(* IEC 61131-3 sources: RL_MAR/experiments/comparison/llm4plc/results/deepseek-ai-DeepSeek-V3.2_20260506_104945/20260506_110207, 3 files *)

(* ---- generated_code_iteration_0.st ---- *)
START_ST
FUNCTION_BLOCK FB_HexDigitAnalyzer
VAR_INPUT
    InputNumber : INT;
END_VAR
VAR_OUTPUT
    Thousands : INT;
    Hundreds : INT;
    Tens : INT;
    Ones : INT;
    Min : INT;
    error : BOOL;
    status : WORD;
END_VAR
VAR
    state : INT;
    prevState : INT;
    tempMin : INT;
    digit1 : INT;
    digit2 : INT;
    digit3 : INT;
    digit4 : INT;
END_VAR

CASE state OF
    0: (* STATE 0: INITIALIZE *)
        Thousands := 0;
        Hundreds := 0;
        Tens := 0;
        Ones := 0;
        Min := 0;
        error := FALSE;
        status := 16#0000;
        state := 1; (* Transition to STATE 1 *)

    1: (* STATE 1: VALIDATE_INPUT *)
        IF (InputNumber >= 0) AND (InputNumber <= 9999) THEN
            error := FALSE;
            status := 16#0000;
            state := 2; (* Valid input, go to digit separation *)
        ELSE
            state := 4; (* Invalid input, go to error handling *)
        END_IF;

    2: (* STATE 2: SEPARATE_DIGITS *)
        Thousands := InputNumber / 1000;
        Hundreds := (InputNumber MOD 1000) / 100;
        Tens := (InputNumber MOD 100) / 10;
        Ones := InputNumber MOD 10;
        state := 3; (* Transition to find minimum *)

    3: (* STATE 3: FIND_MIN_NONZERO_DIGIT *)
        tempMin := 32767; (* Initialize to maximum INT value *)

        digit1 := Thousands;
        IF digit1 <> 0 THEN
            tempMin := minimal(tempMin, digit1);
        END_IF;

        digit2 := Hundreds;
        IF digit2 <> 0 THEN
            tempMin := minimal(tempMin, digit2);
        END_IF;

        digit3 := Tens;
        IF digit3 <> 0 THEN
            tempMin := minimal(tempMin, digit3);
        END_IF;

        digit4 := Ones;
        IF digit4 <> 0 THEN
            tempMin := minimal(tempMin, digit4);
        END_IF;

        IF tempMin = 32767 THEN
            Min := 0; (* All digits were zero *)
        ELSE
            Min := tempMin;
        END_IF;
        state := 0; (* Processing complete, reset for next cycle *)

    4: (* STATE 4: ERROR_HANDLING *)
        Thousands := 0;
        Hundreds := 0;
        Tens := 0;
        Ones := 0;
        Min := 0;
        error := TRUE;
        status := 16#8001;
        state := 0; (* Error handled, reset for next cycle *)

END_CASE;

prevState := state; (* Optional: track previous state if needed for debugging *)

END_FUNCTION_BLOCK
END_ST

(* ---- generated_code_iteration_1.st ---- *)
START_REASON
The validation feedback indicates a CODESYS compiler error: "发现非预期的记号'Min'". This translates to "unexpected token 'Min'". In the context of CODESYS Structured Text, this typically means there is a naming conflict or a reserved word issue. The variable name "Min" might be a reserved keyword or function name in CODESYS (e.g., MIN is a standard function for finding the minimum value). Using "Min" as a variable name can cause a conflict. The solution is to rename the output variable "Min" to something else, such as "MinDigit" or "MinNonZero", to avoid the naming conflict. Additionally, I should ensure that the function "minimal" used in the code is actually "MIN" (the standard CODESYS function). I will rename "Min" to "MinNonZero" and change "minimal" to "MIN". Also, I must maintain the FUNCTION_BLOCK structure and use proper variable declarations.
END_REASON

START_ST
FUNCTION_BLOCK FB_HexDigitAnalyzer
VAR_INPUT
    InputNumber : INT;
END_VAR
VAR_OUTPUT
    Thousands : INT;
    Hundreds : INT;
    Tens : INT;
    Ones : INT;
    MinNonZero : INT;
    error : BOOL;
    status : WORD;
END_VAR
VAR
    state : INT;
    prevState : INT;
    tempMin : INT;
    digit1 : INT;
    digit2 : INT;
    digit3 : INT;
    digit4 : INT;
END_VAR

CASE state OF
    0: (* STATE 0: INITIALIZE *)
        Thousands := 0;
        Hundreds := 0;
        Tens := 0;
        Ones := 0;
        MinNonZero := 0;
        error := FALSE;
        status := 16#0000;
        state := 1; (* Transition to STATE 1 *)

    1: (* STATE 1: VALIDATE_INPUT *)
        IF (InputNumber >= 0) AND (InputNumber <= 9999) THEN
            error := FALSE;
            status := 16#0000;
            state := 2; (* Valid input, go to digit separation *)
        ELSE
            state := 4; (* Invalid input, go to error handling *)
        END_IF;

    2: (* STATE 2: SEPARATE_DIGITS *)
        Thousands := InputNumber / 1000;
        Hundreds := (InputNumber MOD 1000) / 100;
        Tens := (InputNumber MOD 100) / 10;
        Ones := InputNumber MOD 10;
        state := 3; (* Transition to find minimum *)

    3: (* STATE 3: FIND_MIN_NONZERO_DIGIT *)
        tempMin := 32767; (* Initialize to maximum INT value *)

        digit1 := Thousands;
        IF digit1 <> 0 THEN
            tempMin := MIN(tempMin, digit1);
        END_IF;

        digit2 := Hundreds;
        IF digit2 <> 0 THEN
            tempMin := MIN(tempMin, digit2);
        END_IF;

        digit3 := Tens;
        IF digit3 <> 0 THEN
            tempMin := MIN(tempMin, digit3);
        END_IF;

        digit4 := Ones;
        IF digit4 <> 0 THEN
            tempMin := MIN(tempMin, digit4);
        END_IF;

        IF tempMin = 32767 THEN
            MinNonZero := 0; (* All digits were zero *)
        ELSE
            MinNonZero := tempMin;
        END_IF;
        state := 0; (* Processing complete, reset for next cycle *)

    4: (* STATE 4: ERROR_HANDLING *)
        Thousands := 0;
        Hundreds := 0;
        Tens := 0;
        Ones := 0;
        MinNonZero := 0;
        error := TRUE;
        status := 16#8001;
        state := 0; (* Error handled, reset for next cycle *)

END_CASE;

prevState := state; (* Optional: track previous state if needed for debugging *)

END_FUNCTION_BLOCK
END_ST

(* ---- generated_code_iteration_2.st ---- *)
START_REASON
The validation feedback indicates an encoding issue: "'gbk' codec can't decode byte 0xa2 in position 85: illegal multibyte sequence". This suggests there might be a non-ASCII character in the code, possibly in the comments. The byte 0xA2 often corresponds to special characters like the copyright symbol or other non-standard punctuation. Looking at the previous code, I notice comments with parentheses and asterisks, but they appear to be standard ASCII. However, there might be an invisible or special character introduced. To resolve this, I will rewrite the code with simple ASCII comments and ensure no special characters are present. I will also maintain the FUNCTION_BLOCK structure and correct variable declarations as before.
END_REASON

START_ST
FUNCTION_BLOCK FB_HexDigitAnalyzer
VAR_INPUT
    InputNumber : INT;
END_VAR
VAR_OUTPUT
    Thousands : INT;
    Hundreds : INT;
    Tens : INT;
    Ones : INT;
    MinNonZero : INT;
    error : BOOL;
    status : WORD;
END_VAR
VAR
    state : INT;
    prevState : INT;
    tempMin : INT;
    digit1 : INT;
    digit2 : INT;
    digit3 : INT;
    digit4 : INT;
END_VAR

CASE state OF
    0:
        Thousands := 0;
        Hundreds := 0;
        Tens := 0;
        Ones := 0;
        MinNonZero := 0;
        error := FALSE;
        status := 16#0000;
        state := 1;

    1:
        IF (InputNumber >= 0) AND (InputNumber <= 9999) THEN
            error := FALSE;
            status := 16#0000;
            state := 2;
        ELSE
            state := 4;
        END_IF;

    2:
        Thousands := InputNumber / 1000;
        Hundreds := (InputNumber MOD 1000) / 100;
        Tens := (InputNumber MOD 100) / 10;
        Ones := InputNumber MOD 10;
        state := 3;

    3:
        tempMin := 32767;

        digit1 := Thousands;
        IF digit1 <> 0 THEN
            tempMin := MIN(tempMin, digit1);
        END_IF;

        digit2 := Hundreds;
        IF digit2 <> 0 THEN
            tempMin := MIN(tempMin, digit2);
        END_IF;

        digit3 := Tens;
        IF digit3 <> 0 THEN
            tempMin := MIN(tempMin, digit3);
        END_IF;

        digit4 := Ones;
        IF digit4 <> 0 THEN
            tempMin := MIN(tempMin, digit4);
        END_IF;

        IF tempMin = 32767 THEN
            MinNonZero := 0;
        ELSE
            MinNonZero := tempMin;
        END_IF;
        state := 0;

    4:
        Thousands := 0;
        Hundreds := 0;
        Tens := 0;
        Ones := 0;
        MinNonZero := 0;
        error := TRUE;
        status := 16#8001;
        state := 0;

END_CASE;

prevState := state;

END_FUNCTION_BLOCK
END_ST
